TYPE T_TypeID : __UXINT; END_TYPE

(* stored: Version 1.1.0.1
   DUT T_TypeID: Id {b6c9b036-afc1-0bf2-1d7e-809bf7406137} *)
